VAR_GLOBAL PERSISTENT
	OP40_DLY_BEF_MEAS : INT;
	OP40_VERT_SERVO_WORK_POS : REAL;
	OP40_VERT_SERVO_SFE_WORK_POS : REAL;	
END_VAR

(* stored: Version 1.1.0.1, ProductVersion 3.1.4024.11
   GVL OP40_Recipe: Id {c81979df-e8ff-4bd6-b2cf-a0a00a88a59e} *)
